ABB RAPID module: Bandeira_Offs

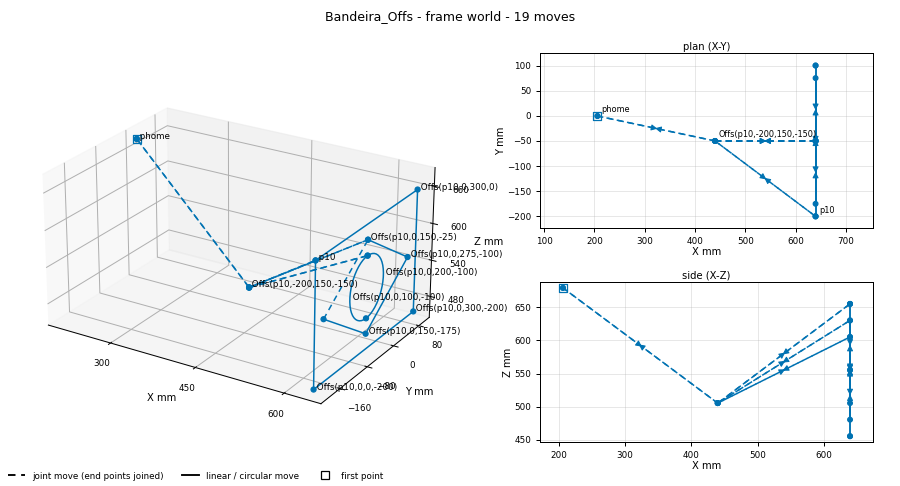
[picture p0: tool path of Bandeira_Offs in frame world, 19 of 19 moves have a stored position in this frame; points joined in program order, loops and branches not executed]
MODULE Module1
    CONST robtarget p10:=[[639.86,-200.00,655.30],[0.500001,3.77523E-06,0.866025,-8.30828E-06],[-1,0,-1,0],[9E+09,9E+09,9E+09,9E+09,9E+09,9E+09]];
    CONST robtarget phome:=[[205.97,-0.43,679.40],[0.500002,-1.72274E-06,0.866024,-2.13775E-07],[-1,0,-1,0],[9E+09,9E+09,9E+09,9E+09,9E+09,9E+09]];
    !***********************************************************
    !
    ! Module:  Module1
    !
    ! Description:
    !   <Insert description here>
    !
    ! Author: Eixo integrativo
    !
    ! Version: 1.0
    !
    !***********************************************************


    !***********************************************************
    !
    ! Procedure main
    !
    !   This is the entry point of your program
    !
    !***********************************************************
    PROC main()
        MoveJ phome, vmax, fine, tool0;
        MoveJ Offs(p10, -200, 150, -150), vmax, fine, tool0;
        !Quadrado
        MoveJ p10, vmax, fine, tool0;
        MoveL Offs(p10, 0, 300, 0), vmax, fine, tool0;
        MoveL Offs(p10, 0, 300, -200), vmax, fine, tool0;
        MoveL Offs(p10, 0, 0, -200), vmax, fine, tool0;
        MoveL p10, vmax, fine, tool0;
        !Retorno
        MoveJ Offs(p10, -200, 150, -150), vmax, fine, tool0;
        !Paralelograma
        MoveJ Offs(p10, 0, 150, -25), vmax, fine, tool0;
        MoveL Offs(p10, 0, 275, -100), vmax, fine, tool0;
        MoveL Offs(p10, 0, 150, -175), vmax, fine, tool0;
        MoveL Offs(p10, 0, 25, -100), vmax, fine, tool0;
        MoveJ Offs(p10, 0, 150, -25), vmax, fine, tool0;
        !Retorno
        MoveJ Offs(p10, -200, 150, -150), vmax, fine, tool0;
        !Circulo
        MoveJ Offs(p10, 0, 150, -50), vmax, fine, tool0;
        MoveC Offs(p10, 0, 200, -100), Offs(p10, 0, 150, -150), vmax, fine, tool0;
        MoveC Offs(p10, 0, 100, -100), Offs(p10, 0, 150, -50), vmax, fine, tool0;
        !phome
        MoveJ Offs(p10, -200, 150, -150), vmax, fine, tool0;
        MoveJ phome, vmax, fine, tool0;
    ENDPROC
ENDMODULE
